Universal Robots PolyScope program: 20240801usb.urp

Program 20240801usb (installation=usb directory=/programs/servoj createdIn=5.13.1 lastSavedIn=5.13.1 robotSerialNumber=20195380017)
Calibrated DH parameters: a=[-0.000005, -0.241897, -0.163857, -0.000004, -0.000042, 0]; d=[0.15198, 4.092034, -18.51686, 14.555458, 0.085328, 0.092191]; alpha=[1.570113, -0.007378, -0.009451, 1.571508, -1.571142, 0]; deltaTheta=[-0.000001, -0.124164, 0.818102, -0.693964, 0.000084, 0]
InitVariablesNode
Robot Program (runOnlyOnce=false)
  MoveJ speed 60 deg/s, acceleration 80 deg/s^2 (useActiveTCP=true) feature=Base
    Waypoint 路点_2: TCP in base x=353.031 y=-286.899 z=146.115 mm, rx=2.8453 ry=-0.8134 rz=0.4989 rad; joints [-21.871, -96.545, -76.602, -76.992, 83.361, -80.357] deg; TCP offset x=-0.542 y=-26.35 z=228.776 mm, rx=0 ry=0 rz=0 rad
  Script: usb = rpc_factory("xmlrpc","http://192.168.1.2:9120/RPC2")
  Script: usb.open()
  Popup Message (haltProgram=false message=Grasp will close... inputType=Text)
  Script: usb.close()
  Script: a=usb.get_target_pose()
  var_3 := p[0,0,0,0,0,0]
  Script: var_3[0] = -a[0]
  Script: var_3[2] = a[2]
  Script: var_3[4] = -a[4]
  Popup Message (haltProgram=false message=Get target pose. inputType=Variable) variable=var_3
  MoveJ speed 60 deg/s, acceleration 80 deg/s^2 (useActiveTCP=true) feature=Base
    Waypoint 路点_1: TCP in base x=219.956 y=-298.93 z=66.445 mm, rx=3.1415 ry=-0.0007 rz=0 rad; joints [-36.966, -107.094, -71.925, -90.964, 89.45, -126.159] deg
  MoveJ speed 30 deg/s, acceleration 60 deg/s^2 (useActiveTCP=true) feature=Base
    var_1 := get_actual_tcp_pose()
    var_2 := pose_trans(var_1, var_3)
    MoveJ speed 60 deg/s, acceleration 80 deg/s^2 (useActiveTCP=true) feature=Base
      Waypoint Variable (Variable): motionParameters(jointSpeed=0.523599 jointAcceleration=1.047198 cartesianSpeed=0.25 cartesianAcceleration=1.2); variable(name=var_2)
  var_4 := var_2
  Script: var_4[2] = var_4[2] - 0.030
  MoveL speed 10 mm/s, acceleration 1200 mm/s^2 (useActiveTCP=true) feature=Base
    Waypoint Variable (Variable): variable(name=var_4)
    Popup Message (haltProgram=false message=Arrived! inputType=Text)
  Script: usb.open()
  Script: var_4[2] = var_4[2] + 0.008
  MoveL speed 10 mm/s, acceleration 1200 mm/s^2 (useActiveTCP=true) feature=Base
    Waypoint Variable (Variable): variable=var_4
  Script: usb.close()
  Script: var_4[2] = var_4[2] - 0.008
  MoveL speed 2 mm/s, acceleration 1000 mm/s^2 (useActiveTCP=true) feature=Base
    Waypoint Variable (Variable): variable=var_4
  Script: usb.open()
  Script: var_4[2] = var_4[2] + 0.04
  MoveL speed 30 mm/s, acceleration 500 mm/s^2 (useActiveTCP=true) feature=Base
    Waypoint Variable (Variable): variable=var_4
